// TIA Portal V19 export
TYPE "LEXCHANGETRAY_typeRoller_toLogisticsReq_B2"
// stored: Access Published
   STRUCT
      inFeedReq : Bool;
      outFeedReq : Bool;   // 请求排料
   END_STRUCT;
END_TYPE
